// TIA Portal V17 export
// export: Created 2023-02-26T22:57:58.9831918Z, ExportSetting WithDefaults, DisplayName Totally Integrated Automation Portal, DisplayVersion V17, DisplayName TIA Portal Openness, DisplayVersion V17, DisplayName TIA Portal Version Control Interface, DisplayVersion V17, DisplayName TIA Portal Test Suite Advanced, DisplayVersion V17, DisplayName STEP 7 Professional, DisplayVersion V17, DisplayName SIMATIC Energy Suite, DisplayVersion V17, DisplayName STEP 7 Safety, DisplayVersion V17, DisplayName WinCC Professional, DisplayVersion V17
FUNCTION_BLOCK "LOG_CountPackage"   // FB4, LAD
{ S7_Optimized_Access := 'TRUE' }
VERSION : 0.1
// stored: AutoNumber true, IsIECCheckEnabled false, IsRetainMemResEnabled false, MemoryReserve 100, SetENOAutomatically false, UDAEnableTagReadback false
   VAR_INPUT
      StartLine : Bool;
      Detector : Bool;
      ResetCountButton : Bool;
   END_VAR
   VAR_OUTPUT
      Quantity : Int;
   END_VAR
   VAR RETAIN
      IEC_Counter_0_Instance { ExternalAccessible := 'False'; ExternalVisible := 'False'; ExternalWritable := 'False'} : CTU_INT;
      N_Detector { S7_SetPoint := 'True'} : Bool;
   END_VAR
   VAR_TEMP   // added for the SCL form of the ladder/FBD networks
      _w1 : Bool;
   END_VAR
BEGIN

REGION Network 1
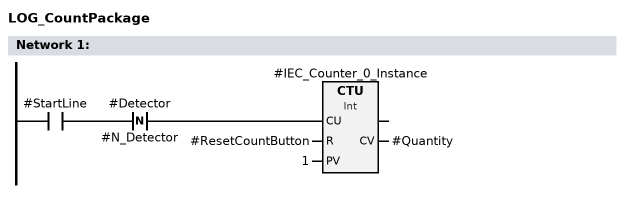
   RUNG wire#powerrail
      Contact( #StartLine )
      N_Contact(operand := #Detector, bit := #N_Detector)
      { S7_Templates := "value_type := Int" } #IEC_Counter_0_Instance.CTU(r := #ResetCountButton, pv := 1, cv => #Quantity)
   END_RUNG
   // the same network as SCL:
   #_w1 := #StartLine AND NOT #Detector AND #N_Detector;   // falling edge of #Detector
   #N_Detector := #Detector;
   #IEC_Counter_0_Instance(CU := #_w1, R := #ResetCountButton, PV := 1, CV => #Quantity);   // CTU
END_REGION
END_FUNCTION_BLOCK
